FUNCTION_BLOCK controller
  (* Standard: 61499-2 *)
  (* Version 0.1, 2017-00-25, hpea485, UOA *)
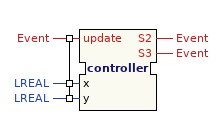
  EVENT_INPUT
    update WITH x, y;
  END_EVENT
  EVENT_OUTPUT
    S2;
    S3;
  END_EVENT
  VAR_INPUT
    x : LREAL;
    y : LREAL;
  END_VAR
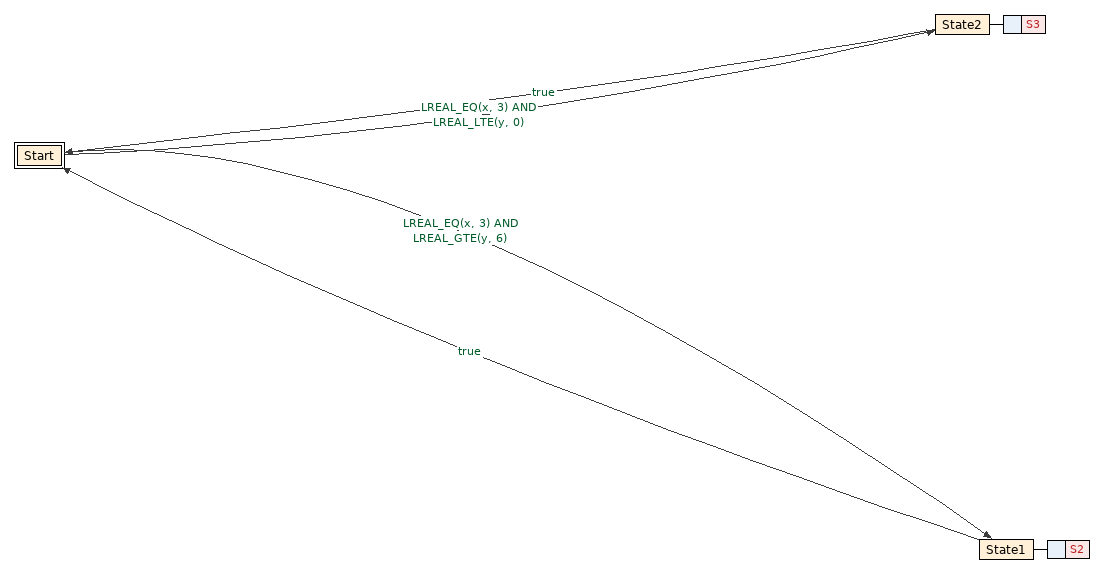
  EC_STATES
    Start;
    State1 : -> S2;
    State2 : -> S3;
  END_STATES
  EC_TRANSITIONS
    Start TO State1 := LREAL_EQ(x, 3) AND LREAL_GTE(y, 6);
    Start TO State2 := LREAL_EQ(x, 3) AND LREAL_LTE(y, 0);
    State1 TO Start := true;
    State2 TO Start := true;
  END_TRANSITIONS
END_FUNCTION_BLOCK
